% RSLogix 500 project digitalFillingStation.RSS, saved by version 8.30.00.16 %
PROJECT "UNTITLED"    % processor: Bul.1763 MicroLogix 1100 Series B %

PROGRAM FILES
  LAD 2   3 rungs
  LAD 3 "I/O"  8 rungs
  LAD 4 "CONTROLS"  8 rungs

DATA FILES
  O0 OUTPUT  4 elements
  I1 INPUT  6 elements
  S2 STATUS  66 elements
  B3 BINARY  2 elements
  T4 TIMER  1 elements
  C5 COUNTER  1 elements
  R6 CONTROL  1 elements
  N7 INTEGER  1 elements
  F8 FLOAT  1 elements

LADDER 2
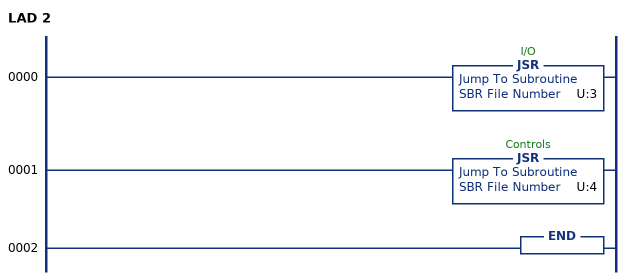
% Rung: 0 %
SOR JSR U:3 EOR
%   U:3  "I/O" %
% Rung: 1 %
SOR JSR U:4 EOR
%   U:4  "Controls" %
% Rung: 2 %
SOR END EOR

LADDER 3 "I/O"
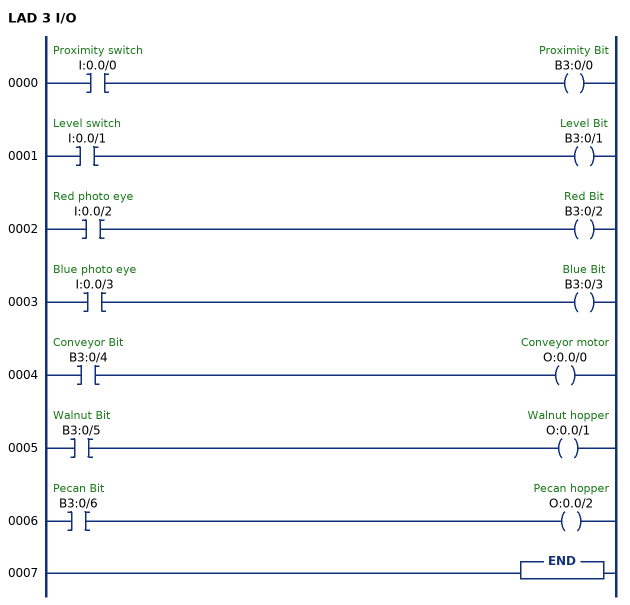
% Rung: 0 %
SOR XIC I:0.0/0 OTE B3:0/0 EOR
%   I:0.0/0  "Proximity switch" %
%   B3:0/0  "Proximity Bit" %
% Rung: 1 %
SOR XIC I:0.0/1 OTE B3:0/1 EOR
%   I:0.0/1  "Level switch" %
%   B3:0/1  "Level Bit" %
% Rung: 2 %
SOR XIC I:0.0/2 OTE B3:0/2 EOR
%   I:0.0/2  "Red photo eye" %
%   B3:0/2  "Red Bit" %
% Rung: 3 %
SOR XIC I:0.0/3 OTE B3:0/3 EOR
%   I:0.0/3  "Blue photo eye" %
%   B3:0/3  "Blue Bit" %
% Rung: 4 %
SOR XIC B3:0/4 OTE O:0.0/0 EOR
%   B3:0/4  "Conveyor Bit" %
%   O:0.0/0  "Conveyor motor" %
% Rung: 5 %
SOR XIC B3:0/5 OTE O:0.0/1 EOR
%   B3:0/5  "Walnut Bit" %
%   O:0.0/1  "Walnut hopper" %
% Rung: 6 %
SOR XIC B3:0/6 OTE O:0.0/2 EOR
%   B3:0/6  "Pecan Bit" %
%   O:0.0/2  "Pecan hopper" %
% Rung: 7 %
SOR END EOR

LADDER 4 "CONTROLS"
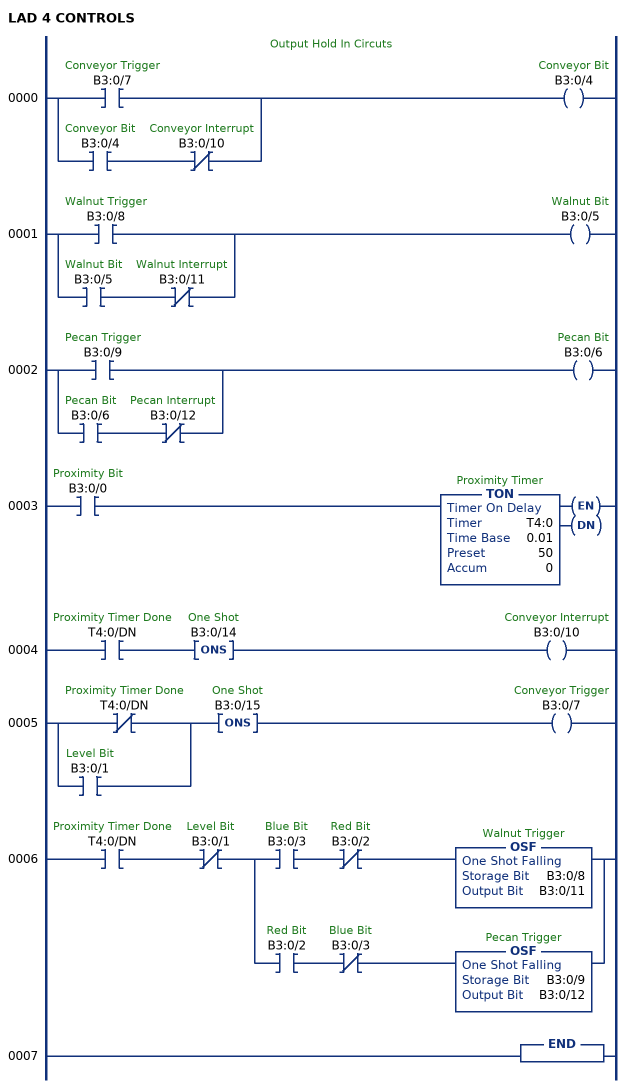
% Rung: 0 %
% Output Hold In Circuts %
SOR BST XIC B3:0/7 NXB XIC B3:0/4 XIO B3:0/10 BND OTE B3:0/4 EOR
%   B3:0/7  "Conveyor Trigger" %
%   B3:0/4  "Conveyor Bit" %
%   B3:0/10  "Conveyor Interrupt" %
% Rung: 1 %
SOR BST XIC B3:0/8 NXB XIC B3:0/5 XIO B3:0/11 BND OTE B3:0/5 EOR
%   B3:0/8  "Walnut Trigger" %
%   B3:0/5  "Walnut Bit" %
%   B3:0/11  "Walnut Interrupt" %
% Rung: 2 %
SOR BST XIC B3:0/9 NXB XIC B3:0/6 XIO B3:0/12 BND OTE B3:0/6 EOR
%   B3:0/9  "Pecan Trigger" %
%   B3:0/6  "Pecan Bit" %
%   B3:0/12  "Pecan Interrupt" %
% Rung: 3 %
SOR XIC B3:0/0 TON T4:0 0.01 50 0 EOR
%   B3:0/0  "Proximity Bit" %
%   T4:0  "Proximity Timer" %
% Rung: 4 %
SOR XIC T4:0/DN ONS B3:0/14 OTE B3:0/10 EOR
%   T4:0/DN  "Proximity Timer Done" %
%   B3:0/14  "One Shot" %
%   B3:0/10  "Conveyor Interrupt" %
% Rung: 5 %
SOR BST XIO T4:0/DN NXB XIC B3:0/1 BND ONS B3:0/15 OTE B3:0/7 EOR
%   T4:0/DN  "Proximity Timer Done" %
%   B3:0/1  "Level Bit" %
%   B3:0/15  "One Shot" %
%   B3:0/7  "Conveyor Trigger" %
% Rung: 6 %
SOR XIC T4:0/DN XIO B3:0/1 BST XIC B3:0/3 XIO B3:0/2 OSF B3:0/8 B3:0/11 NXB XIC B3:0/2 XIO B3:0/3 OSF B3:0/9 B3:0/12 BND EOR
%   T4:0/DN  "Proximity Timer Done" %
%   B3:0/1  "Level Bit" %
%   B3:0/3  "Blue Bit" %
%   B3:0/2  "Red Bit" %
%   B3:0/8  "Walnut Trigger" %
%   B3:0/11  "Walnut Interrupt" %
%   B3:0/9  "Pecan Trigger" %
%   B3:0/12  "Pecan Interrupt" %
% Rung: 7 %
SOR END EOR

OTHER DOCUMENTED ADDRESSES
  B3:0/13  "Hopper Selector"
  B3:1/0  "One Shot"
  B3:1/1  "One Shot"
  B3:10  "Conveyor Interrupt"
  PFILE:3  "I/O"

DATA TABLE (non-zero values as saved)
DATA T4
% .PRE .ACC %
% T4:0 % 50 0
